ABB RAPID module: 93bc2229-db1b-41b8-8230-48410be7e35f-Module1.mod

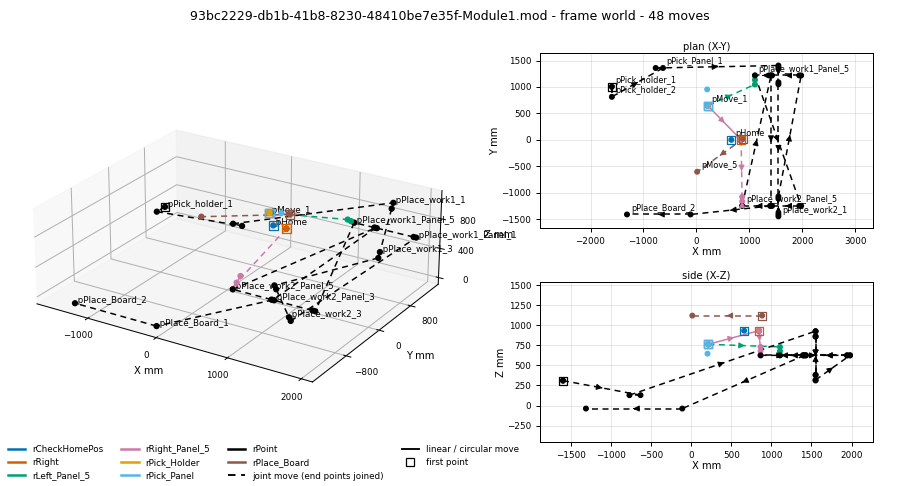
[picture p0: tool path of 93bc2229-db1b-41b8-8230-48410be7e35f-Module1.mod in frame world, 48 of 79 moves have a stored position in this frame; points joined in program order, loops and branches not executed]
MODULE Module1
    PERS tooldata Tool_Vacuum:=[TRUE,[[0,0.098,155.795],[1,0,0,0]],[5,[0,0,50],[1,0,0,0],0,0,0]];
	TASK PERS wobjdata Wobj_materials:=[FALSE,TRUE,"",[[-2196.81,858.538,-168],[1,0,0,0]],[[0,0,0],[1,0,0,0]]];
	TASK PERS wobjdata Wobj_Board:=[FALSE,TRUE,"",[[-2051.58,-1907.53,-168],[1,0,0,0]],[[0,0,0],[1,0,0,0]]];
	TASK PERS wobjdata Wobj_Left:=[FALSE,TRUE,"",[[802.356,885.126,-138],[0.872954,0.487803,0,0]],[[0,0,0],[1,0,0,0]]];
	TASK PERS wobjdata Wobj_Right:=[FALSE,TRUE,"",[[802.356,-1714.87,1162],[0.872954,-0.487803,0,0]],[[0,0,0],[1,0,0,0]]];
    PERS robtarget pHome:=[[661.17,-0.00,932.98],[3.16101E-08,-0.707107,-0.707107,-7.01508E-10],[-1,0,0,0],[9E+09,9E+09,9E+09,9E+09,9E+09,9E+09]];
    PERS robtarget pPick_holder_1:=[[600.00,145.65,477.91],[4.68845E-08,1.19209E-07,1,-2.94814E-08],[1,0,1,0],[9E+09,9E+09,9E+09,9E+09,9E+09,9E+09]];
    PERS robtarget pPick_holder_2:=[[600.00,-45.54,478.84],[7.08134E-08,4.45843E-09,1,-4.04558E-08],[1,0,1,0],[9E+09,9E+09,9E+09,9E+09,9E+09,9E+09]];
    PERS robtarget pPick_Panel_1:=[[1566.56,500.00,297.53],[2.60305E-09,0.707107,0.707107,-1.31181E-08],[1,0,2,0],[9E+09,9E+09,9E+09,9E+09,9E+09,9E+09]];
    PERS robtarget pPick_Panel_2:=[[1428.44,500.00,297.53],[3.82813E-09,0.707107,0.707107,-1.22165E-08],[1,0,2,0],[9E+09,9E+09,9E+09,9E+09,9E+09,9E+09]];
    PERS robtarget pPick_Holder_Move1{4,10}:=[[[[600,145.65,477.91],[4.68845E-8,1.19209E-7,1,-2.94814E-8],[1,0,1,0],[9E+9,9E+9,9E+9,9E+9,9E+9,9E+9]],[[600,245.65,477.91],[4.68845E-8,1.19209E-7,1,-2.94814E-8],[1,0,1,0],[9E+9,9E+9,9E+9,9E+9,9E+9,9E+9]],[[600,345.65,477.91],[4.68845E-8,1.19209E-7,1,-2.94814E-8],[1,0,1,0],[9E+9,9E+9,9E+9,9E+9,9E+9,9E+9]],[[600,445.65,477.91],[4.68845E-8,1.19209E-7,1,-2.94814E-8],[1,0,1,0],[9E+9,9E+9,9E+9,9E+9,9E+9,9E+9]],[[600,545.65,477.91],[4.68845E-8,1.19209E-7,1,-2.94814E-8],[1,0,1,0],[9E+9,9E+9,9E+9,9E+9,9E+9,9E+9]],[[600,645.65,477.91],[4.68845E-8,1.19209E-7,1,-2.94814E-8],[1,0,1,0],[9E+9,9E+9,9E+9,9E+9,9E+9,9E+9]],[[600,745.65,477.91],[4.68845E-8,1.19209E-7,1,-2.94814E-8],[1,0,1,0],[9E+9,9E+9,9E+9,9E+9,9E+9,9E+9]],[[600,845.65,477.91],[4.68845E-8,1.19209E-7,1,-2.94814E-8],[1,0,1,0],[9E+9,9E+9,9E+9,9E+9,9E+9,9E+9]],[[600,945.65,477.91],[4.68845E-8,1.19209E-7,1,-2.94814E-8],[1,0,1,0],[9E+9,9E+9,9E+9,9E+9,9E+9,9E+9]],[[600,1045.65,477.91],[4.68845E-8,1.19209E-7,1,-2.94814E-8],[1,0,1,0],[9E+9,9E+9,9E+9,9E+9,9E+9,9E+9]]],[[[600,145.65,357.91],[4.68845E-8,1.19209E-7,1,-2.94814E-8],[1,0,1,0],[9E+9,9E+9,9E+9,9E+9,9E+9,9E+9]],[[600,245.65,357.91],[4.68845E-8,1.19209E-7,1,-2.94814E-8],[1,0,1,0],[9E+9,9E+9,9E+9,9E+9,9E+9,9E+9]],[[600,345.65,357.91],[4.68845E-8,1.19209E-7,1,-2.94814E-8],[1,0,1,0],[9E+9,9E+9,9E+9,9E+9,9E+9,9E+9]],[[600,445.65,357.91],[4.68845E-8,1.19209E-7,1,-2.94814E-8],[1,0,1,0],[9E+9,9E+9,9E+9,9E+9,9E+9,9E+9]],[[600,545.65,357.91],[4.68845E-8,1.19209E-7,1,-2.94814E-8],[1,0,1,0],[9E+9,9E+9,9E+9,9E+9,9E+9,9E+9]],[[600,645.65,357.91],[4.68845E-8,1.19209E-7,1,-2.94814E-8],[1,0,1,0],[9E+9,9E+9,9E+9,9E+9,9E+9,9E+9]],[[600,745.65,357.91],[4.68845E-8,1.19209E-7,1,-2.94814E-8],[1,0,1,0],[9E+9,9E+9,9E+9,9E+9,9E+9,9E+9]],[[600,845.65,357.91],[4.68845E-8,1.19209E-7,1,-2.94814E-8],[1,0,1,0],[9E+9,9E+9,9E+9,9E+9,9E+9,9E+9]],[[600,945.65,357.91],[4.68845E-8,1.19209E-7,1,-2.94814E-8],[1,0,1,0],[9E+9,9E+9,9E+9,9E+9,9E+9,9E+9]],[[600,1045.65,357.91],[4.68845E-8,1.19209E-7,1,-2.94814E-8],[1,0,1,0],[9E+9,9E+9,9E+9,9E+9,9E+9,9E+9]]],[[[600,145.65,237.91],[4.68845E-8,1.19209E-7,1,-2.94814E-8],[1,0,1,0],[9E+9,9E+9,9E+9,9E+9,9E+9,9E+9]],[[600,245.65,237.91],[4.68845E-8,1.19209E-7,1,-2.94814E-8],[1,0,1,0],[9E+9,9E+9,9E+9,9E+9,9E+9,9E+9]],[[600,345.65,237.91],[4.68845E-8,1.19209E-7,1,-2.94814E-8],[1,0,1,0],[9E+9,9E+9,9E+9,9E+9,9E+9,9E+9]],[[600,445.65,237.91],[4.68845E-8,1.19209E-7,1,-2.94814E-8],[1,0,1,0],[9E+9,9E+9,9E+9,9E+9,9E+9,9E+9]],[[600,545.65,237.91],[4.68845E-8,1.19209E-7,1,-2.94814E-8],[1,0,1,0],[9E+9,9E+9,9E+9,9E+9,9E+9,9E+9]],[[600,645.65,237.91],[4.68845E-8,1.19209E-7,1,-2.94814E-8],[1,0,1,0],[9E+9,9E+9,9E+9,9E+9,9E+9,9E+9]],[[600,745.65,237.91],[4.68845E-8,1.19209E-7,1,-2.94814E-8],[1,0,1,0],[9E+9,9E+9,9E+9,9E+9,9E+9,9E+9]],[[600,845.65,237.91],[4.68845E-8,1.19209E-7,1,-2.94814E-8],[1,0,1,0],[9E+9,9E+9,9E+9,9E+9,9E+9,9E+9]],[[600,945.65,237.91],[4.68845E-8,1.19209E-7,1,-2.94814E-8],[1,0,1,0],[9E+9,9E+9,9E+9,9E+9,9E+9,9E+9]],[[600,1045.65,237.91],[4.68845E-8,1.19209E-7,1,-2.94814E-8],[1,0,1,0],[9E+9,9E+9,9E+9,9E+9,9E+9,9E+9]]],[[[600,145.65,117.91],[4.68845E-8,1.19209E-7,1,-2.94814E-8],[1,0,1,0],[9E+9,9E+9,9E+9,9E+9,9E+9,9E+9]],[[600,245.65,117.91],[4.68845E-8,1.19209E-7,1,-2.94814E-8],[1,0,1,0],[9E+9,9E+9,9E+9,9E+9,9E+9,9E+9]],[[600,345.65,117.91],[4.68845E-8,1.19209E-7,1,-2.94814E-8],[1,0,1,0],[9E+9,9E+9,9E+9,9E+9,9E+9,9E+9]],[[600,445.65,117.91],[4.68845E-8,1.19209E-7,1,-2.94814E-8],[1,0,1,0],[9E+9,9E+9,9E+9,9E+9,9E+9,9E+9]],[[600,545.65,117.91],[4.68845E-8,1.19209E-7,1,-2.94814E-8],[1,0,1,0],[9E+9,9E+9,9E+9,9E+9,9E+9,9E+9]],[[600,645.65,117.91],[4.68845E-8,1.19209E-7,1,-2.94814E-8],[1,0,1,0],[9E+9,9E+9,9E+9,9E+9,9E+9,9E+9]],[[600,745.65,117.91],[4.68845E-8,1.19209E-7,1,-2.94814E-8],[1,0,1,0],[9E+9,9E+9,9E+9,9E+9,9E+9,9E+9]],[[600,845.65,117.91],[4.68845E-8,1.19209E-7,1,-2.94814E-8],[1,0,1,0],[9E+9,9E+9,9E+9,9E+9,9E+9,9E+9]],[[600,945.65,117.91],[4.68845E-8,1.19209E-7,1,-2.94814E-8],[1,0,1,0],[9E+9,9E+9,9E+9,9E+9,9E+9,9E+9]],[[600,1045.65,117.91],[4.68845E-8,1.19209E-7,1,-2.94814E-8],[1,0,1,0],[9E+9,9E+9,9E+9,9E+9,9E+9,9E+9]]]];
    PERS robtarget pPick_Holder_Move2{4,10}:=[[[[600,-45.54,478.84],[7.08134E-8,4.45843E-9,1,-4.04558E-8],[1,0,1,0],[9E+9,9E+9,9E+9,9E+9,9E+9,9E+9]],[[600,54.46,478.84],[7.08134E-8,4.45843E-9,1,-4.04558E-8],[1,0,1,0],[9E+9,9E+9,9E+9,9E+9,9E+9,9E+9]],[[600,154.46,478.84],[7.08134E-8,4.45843E-9,1,-4.04558E-8],[1,0,1,0],[9E+9,9E+9,9E+9,9E+9,9E+9,9E+9]],[[600,254.46,478.84],[7.08134E-8,4.45843E-9,1,-4.04558E-8],[1,0,1,0],[9E+9,9E+9,9E+9,9E+9,9E+9,9E+9]],[[600,354.46,478.84],[7.08134E-8,4.45843E-9,1,-4.04558E-8],[1,0,1,0],[9E+9,9E+9,9E+9,9E+9,9E+9,9E+9]],[[600,454.46,478.84],[7.08134E-8,4.45843E-9,1,-4.04558E-8],[1,0,1,0],[9E+9,9E+9,9E+9,9E+9,9E+9,9E+9]],[[600,554.46,478.84],[7.08134E-8,4.45843E-9,1,-4.04558E-8],[1,0,1,0],[9E+9,9E+9,9E+9,9E+9,9E+9,9E+9]],[[600,654.46,478.84],[7.08134E-8,4.45843E-9,1,-4.04558E-8],[1,0,1,0],[9E+9,9E+9,9E+9,9E+9,9E+9,9E+9]],[[600,754.46,478.84],[7.08134E-8,4.45843E-9,1,-4.04558E-8],[1,0,1,0],[9E+9,9E+9,9E+9,9E+9,9E+9,9E+9]],[[600,854.46,478.84],[7.08134E-8,4.45843E-9,1,-4.04558E-8],[1,0,1,0],[9E+9,9E+9,9E+9,9E+9,9E+9,9E+9]]],[[[600,-45.54,358.84],[7.08134E-8,4.45843E-9,1,-4.04558E-8],[1,0,1,0],[9E+9,9E+9,9E+9,9E+9,9E+9,9E+9]],[[600,54.46,358.84],[7.08134E-8,4.45843E-9,1,-4.04558E-8],[1,0,1,0],[9E+9,9E+9,9E+9,9E+9,9E+9,9E+9]],[[600,154.46,358.84],[7.08134E-8,4.45843E-9,1,-4.04558E-8],[1,0,1,0],[9E+9,9E+9,9E+9,9E+9,9E+9,9E+9]],[[600,254.46,358.84],[7.08134E-8,4.45843E-9,1,-4.04558E-8],[1,0,1,0],[9E+9,9E+9,9E+9,9E+9,9E+9,9E+9]],[[600,354.46,358.84],[7.08134E-8,4.45843E-9,1,-4.04558E-8],[1,0,1,0],[9E+9,9E+9,9E+9,9E+9,9E+9,9E+9]],[[600,454.46,358.84],[7.08134E-8,4.45843E-9,1,-4.04558E-8],[1,0,1,0],[9E+9,9E+9,9E+9,9E+9,9E+9,9E+9]],[[600,554.46,358.84],[7.08134E-8,4.45843E-9,1,-4.04558E-8],[1,0,1,0],[9E+9,9E+9,9E+9,9E+9,9E+9,9E+9]],[[600,654.46,358.84],[7.08134E-8,4.45843E-9,1,-4.04558E-8],[1,0,1,0],[9E+9,9E+9,9E+9,9E+9,9E+9,9E+9]],[[600,754.46,358.84],[7.08134E-8,4.45843E-9,1,-4.04558E-8],[1,0,1,0],[9E+9,9E+9,9E+9,9E+9,9E+9,9E+9]],[[600,854.46,358.84],[7.08134E-8,4.45843E-9,1,-4.04558E-8],[1,0,1,0],[9E+9,9E+9,9E+9,9E+9,9E+9,9E+9]]],[[[600,-45.54,238.84],[7.08134E-8,4.45843E-9,1,-4.04558E-8],[1,0,1,0],[9E+9,9E+9,9E+9,9E+9,9E+9,9E+9]],[[600,54.46,238.84],[7.08134E-8,4.45843E-9,1,-4.04558E-8],[1,0,1,0],[9E+9,9E+9,9E+9,9E+9,9E+9,9E+9]],[[600,154.46,238.84],[7.08134E-8,4.45843E-9,1,-4.04558E-8],[1,0,1,0],[9E+9,9E+9,9E+9,9E+9,9E+9,9E+9]],[[600,254.46,238.84],[7.08134E-8,4.45843E-9,1,-4.04558E-8],[1,0,1,0],[9E+9,9E+9,9E+9,9E+9,9E+9,9E+9]],[[600,354.46,238.84],[7.08134E-8,4.45843E-9,1,-4.04558E-8],[1,0,1,0],[9E+9,9E+9,9E+9,9E+9,9E+9,9E+9]],[[600,454.46,238.84],[7.08134E-8,4.45843E-9,1,-4.04558E-8],[1,0,1,0],[9E+9,9E+9,9E+9,9E+9,9E+9,9E+9]],[[600,554.46,238.84],[7.08134E-8,4.45843E-9,1,-4.04558E-8],[1,0,1,0],[9E+9,9E+9,9E+9,9E+9,9E+9,9E+9]],[[600,654.46,238.84],[7.08134E-8,4.45843E-9,1,-4.04558E-8],[1,0,1,0],[9E+9,9E+9,9E+9,9E+9,9E+9,9E+9]],[[600,754.46,238.84],[7.08134E-8,4.45843E-9,1,-4.04558E-8],[1,0,1,0],[9E+9,9E+9,9E+9,9E+9,9E+9,9E+9]],[[600,854.46,238.84],[7.08134E-8,4.45843E-9,1,-4.04558E-8],[1,0,1,0],[9E+9,9E+9,9E+9,9E+9,9E+9,9E+9]]],[[[600,-45.54,118.84],[7.08134E-8,4.45843E-9,1,-4.04558E-8],[1,0,1,0],[9E+9,9E+9,9E+9,9E+9,9E+9,9E+9]],[[600,54.46,118.84],[7.08134E-8,4.45843E-9,1,-4.04558E-8],[1,0,1,0],[9E+9,9E+9,9E+9,9E+9,9E+9,9E+9]],[[600,154.46,118.84],[7.08134E-8,4.45843E-9,1,-4.04558E-8],[1,0,1,0],[9E+9,9E+9,9E+9,9E+9,9E+9,9E+9]],[[600,254.46,118.84],[7.08134E-8,4.45843E-9,1,-4.04558E-8],[1,0,1,0],[9E+9,9E+9,9E+9,9E+9,9E+9,9E+9]],[[600,354.46,118.84],[7.08134E-8,4.45843E-9,1,-4.04558E-8],[1,0,1,0],[9E+9,9E+9,9E+9,9E+9,9E+9,9E+9]],[[600,454.46,118.84],[7.08134E-8,4.45843E-9,1,-4.04558E-8],[1,0,1,0],[9E+9,9E+9,9E+9,9E+9,9E+9,9E+9]],[[600,554.46,118.84],[7.08134E-8,4.45843E-9,1,-4.04558E-8],[1,0,1,0],[9E+9,9E+9,9E+9,9E+9,9E+9,9E+9]],[[600,654.46,118.84],[7.08134E-8,4.45843E-9,1,-4.04558E-8],[1,0,1,0],[9E+9,9E+9,9E+9,9E+9,9E+9,9E+9]],[[600,754.46,118.84],[7.08134E-8,4.45843E-9,1,-4.04558E-8],[1,0,1,0],[9E+9,9E+9,9E+9,9E+9,9E+9,9E+9]],[[600,854.46,118.84],[7.08134E-8,4.45843E-9,1,-4.04558E-8],[1,0,1,0],[9E+9,9E+9,9E+9,9E+9,9E+9,9E+9]]]];
    PERS robtarget pPick_Panel_Move1{20,5}:=[[[[1566.56,500,297.53],[2.60305E-9,0.707107,0.707107,-1.31181E-8],[1,0,2,0],[9E+9,9E+9,9E+9,9E+9,9E+9,9E+9]],[[1766.56,500,297.53],[2.60305E-9,0.707107,0.707107,-1.31181E-8],[1,0,2,0],[9E+9,9E+9,9E+9,9E+9,9E+9,9E+9]],[[1966.56,500,297.53],[2.60305E-9,0.707107,0.707107,-1.31181E-8],[1,0,2,0],[9E+9,9E+9,9E+9,9E+9,9E+9,9E+9]],[[2166.56,500,297.53],[2.60305E-9,0.707107,0.707107,-1.31181E-8],[1,0,2,0],[9E+9,9E+9,9E+9,9E+9,9E+9,9E+9]],[[2366.56,500,297.53],[2.60305E-9,0.707107,0.707107,-1.31181E-8],[1,0,2,0],[9E+9,9E+9,9E+9,9E+9,9E+9,9E+9]]],[[[1566.56,500,282.53],[2.60305E-9,0.707107,0.707107,-1.31181E-8],[1,0,2,0],[9E+9,9E+9,9E+9,9E+9,9E+9,9E+9]],[[1766.56,500,282.53],[2.60305E-9,0.707107,0.707107,-1.31181E-8],[1,0,2,0],[9E+9,9E+9,9E+9,9E+9,9E+9,9E+9]],[[1966.56,500,282.53],[2.60305E-9,0.707107,0.707107,-1.31181E-8],[1,0,2,0],[9E+9,9E+9,9E+9,9E+9,9E+9,9E+9]],[[2166.56,500,282.53],[2.60305E-9,0.707107,0.707107,-1.31181E-8],[1,0,2,0],[9E+9,9E+9,9E+9,9E+9,9E+9,9E+9]],[[2366.56,500,282.53],[2.60305E-9,0.707107,0.707107,-1.31181E-8],[1,0,2,0],[9E+9,9E+9,9E+9,9E+9,9E+9,9E+9]]],[[[1566.56,500,267.53],[2.60305E-9,0.707107,0.707107,-1.31181E-8],[1,0,2,0],[9E+9,9E+9,9E+9,9E+9,9E+9,9E+9]],[[1766.56,500,267.53],[2.60305E-9,0.707107,0.707107,-1.31181E-8],[1,0,2,0],[9E+9,9E+9,9E+9,9E+9,9E+9,9E+9]],[[1966.56,500,267.53],[2.60305E-9,0.707107,0.707107,-1.31181E-8],[1,0,2,0],[9E+9,9E+9,9E+9,9E+9,9E+9,9E+9]],[[2166.56,500,267.53],[2.60305E-9,0.707107,0.707107,-1.31181E-8],[1,0,2,0],[9E+9,9E+9,9E+9,9E+9,9E+9,9E+9]],[[2366.56,500,267.53],[2.60305E-9,0.707107,0.707107,-1.31181E-8],[1,0,2,0],[9E+9,9E+9,9E+9,9E+9,9E+9,9E+9]]],[[[1566.56,500,252.53],[2.60305E-9,0.707107,0.707107,-1.31181E-8],[1,0,2,0],[9E+9,9E+9,9E+9,9E+9,9E+9,9E+9]],[[1766.56,500,252.53],[2.60305E-9,0.707107,0.707107,-1.31181E-8],[1,0,2,0],[9E+9,9E+9,9E+9,9E+9,9E+9,9E+9]],[[1966.56,500,252.53],[2.60305E-9,0.707107,0.707107,-1.31181E-8],[1,0,2,0],[9E+9,9E+9,9E+9,9E+9,9E+9,9E+9]],[[2166.56,500,252.53],[2.60305E-9,0.707107,0.707107,-1.31181E-8],[1,0,2,0],[9E+9,9E+9,9E+9,9E+9,9E+9,9E+9]],[[2366.56,500,252.53],[2.60305E-9,0.707107,0.707107,-1.31181E-8],[1,0,2,0],[9E+9,9E+9,9E+9,9E+9,9E+9,9E+9]]],[[[1566.56,500,237.53],[2.60305E-9,0.707107,0.707107,-1.31181E-8],[1,0,2,0],[9E+9,9E+9,9E+9,9E+9,9E+9,9E+9]],[[1766.56,500,237.53],[2.60305E-9,0.707107,0.707107,-1.31181E-8],[1,0,2,0],[9E+9,9E+9,9E+9,9E+9,9E+9,9E+9]],[[1966.56,500,237.53],[2.60305E-9,0.707107,0.707107,-1.31181E-8],[1,0,2,0],[9E+9,9E+9,9E+9,9E+9,9E+9,9E+9]],[[2166.56,500,237.53],[2.60305E-9,0.707107,0.707107,-1.31181E-8],[1,0,2,0],[9E+9,9E+9,9E+9,9E+9,9E+9,9E+9]],[[2366.56,500,237.53],[2.60305E-9,0.707107,0.707107,-1.31181E-8],[1,0,2,0],[9E+9,9E+9,9E+9,9E+9,9E+9,9E+9]]],[[[1566.56,500,222.53],[2.60305E-9,0.707107,0.707107,-1.31181E-8],[1,0,2,0],[9E+9,9E+9,9E+9,9E+9,9E+9,9E+9]],[[1766.56,500,222.53],[2.60305E-9,0.707107,0.707107,-1.31181E-8],[1,0,2,0],[9E+9,9E+9,9E+9,9E+9,9E+9,9E+9]],[[1966.56,500,222.53],[2.60305E-9,0.707107,0.707107,-1.31181E-8],[1,0,2,0],[9E+9,9E+9,9E+9,9E+9,9E+9,9E+9]],[[2166.56,500,222.53],[2.60305E-9,0.707107,0.707107,-1.31181E-8],[1,0,2,0],[9E+9,9E+9,9E+9,9E+9,9E+9,9E+9]],[[2366.56,500,222.53],[2.60305E-9,0.707107,0.707107,-1.31181E-8],[1,0,2,0],[9E+9,9E+9,9E+9,9E+9,9E+9,9E+9]]],[[[1566.56,500,207.53],[2.60305E-9,0.707107,0.707107,-1.31181E-8],[1,0,2,0],[9E+9,9E+9,9E+9,9E+9,9E+9,9E+9]],[[1766.56,500,207.53],[2.60305E-9,0.707107,0.707107,-1.31181E-8],[1,0,2,0],[9E+9,9E+9,9E+9,9E+9,9E+9,9E+9]],[[1966.56,500,207.53],[2.60305E-9,0.707107,0.707107,-1.31181E-8],[1,0,2,0],[9E+9,9E+9,9E+9,9E+9,9E+9,9E+9]],[[2166.56,500,207.53],[2.60305E-9,0.707107,0.707107,-1.31181E-8],[1,0,2,0],[9E+9,9E+9,9E+9,9E+9,9E+9,9E+9]],[[2366.56,500,207.53],[2.60305E-9,0.707107,0.707107,-1.31181E-8],[1,0,2,0],[9E+9,9E+9,9E+9,9E+9,9E+9,9E+9]]],[[[1566.56,500,192.53],[2.60305E-9,0.707107,0.707107,-1.31181E-8],[1,0,2,0],[9E+9,9E+9,9E+9,9E+9,9E+9,9E+9]],[[1766.56,500,192.53],[2.60305E-9,0.707107,0.707107,-1.31181E-8],[1,0,2,0],[9E+9,9E+9,9E+9,9E+9,9E+9,9E+9]],[[1966.56,500,192.53],[2.60305E-9,0.707107,0.707107,-1.31181E-8],[1,0,2,0],[9E+9,9E+9,9E+9,9E+9,9E+9,9E+9]],[[2166.56,500,192.53],[2.60305E-9,0.707107,0.707107,-1.31181E-8],[1,0,2,0],[9E+9,9E+9,9E+9,9E+9,9E+9,9E+9]],[[2366.56,500,192.53],[2.60305E-9,0.707107,0.707107,-1.31181E-8],[1,0,2,0],[9E+9,9E+9,9E+9,9E+9,9E+9,9E+9]]],[[[1566.56,500,177.53],[2.60305E-9,0.707107,0.707107,-1.31181E-8],[1,0,2,0],[9E+9,9E+9,9E+9,9E+9,9E+9,9E+9]],[[1766.56,500,177.53],[2.60305E-9,0.707107,0.707107,-1.31181E-8],[1,0,2,0],[9E+9,9E+9,9E+9,9E+9,9E+9,9E+9]],[[1966.56,500,177.53],[2.60305E-9,0.707107,0.707107,-1.31181E-8],[1,0,2,0],[9E+9,9E+9,9E+9,9E+9,9E+9,9E+9]],[[2166.56,500,177.53],[2.60305E-9,0.707107,0.707107,-1.31181E-8],[1,0,2,0],[9E+9,9E+9,9E+9,9E+9,9E+9,9E+9]],[[2366.56,500,177.53],[2.60305E-9,0.707107,0.707107,-1.31181E-8],[1,0,2,0],[9E+9,9E+9,9E+9,9E+9,9E+9,9E+9]]],[[[1566.56,500,162.53],[2.60305E-9,0.707107,0.707107,-1.31181E-8],[1,0,2,0],[9E+9,9E+9,9E+9,9E+9,9E+9,9E+9]],[[1766.56,500,162.53],[2.60305E-9,0.707107,0.707107,-1.31181E-8],[1,0,2,0],[9E+9,9E+9,9E+9,9E+9,9E+9,9E+9]],[[1966.56,500,162.53],[2.60305E-9,0.707107,0.707107,-1.31181E-8],[1,0,2,0],[9E+9,9E+9,9E+9,9E+9,9E+9,9E+9]],[[2166.56,500,162.53],[2.60305E-9,0.707107,0.707107,-1.31181E-8],[1,0,2,0],[9E+9,9E+9,9E+9,9E+9,9E+9,9E+9]],[[2366.56,500,162.53],[2.60305E-9,0.707107,0.707107,-1.31181E-8],[1,0,2,0],[9E+9,9E+9,9E+9,9E+9,9E+9,9E+9]]],[[[1566.56,500,147.53],[2.60305E-9,0.707107,0.707107,-1.31181E-8],[1,0,2,0],[9E+9,9E+9,9E+9,9E+9,9E+9,9E+9]],[[1766.56,500,147.53],[2.60305E-9,0.707107,0.707107,-1.31181E-8],[1,0,2,0],[9E+9,9E+9,9E+9,9E+9,9E+9,9E+9]],[[1966.56,500,147.53],[2.60305E-9,0.707107,0.707107,-1.31181E-8],[1,0,2,0],[9E+9,9E+9,9E+9,9E+9,9E+9,9E+9]],[[2166.56,500,147.53],[2.60305E-9,0.707107,0.707107,-1.31181E-8],[1,0,2,0],[9E+9,9E+9,9E+9,9E+9,9E+9,9E+9]],[[2366.56,500,147.53],[2.60305E-9,0.707107,0.707107,-1.31181E-8],[1,0,2,0],[9E+9,9E+9,9E+9,9E+9,9E+9,9E+9]]],[[[1566.56,500,132.53],[2.60305E-9,0.707107,0.707107,-1.31181E-8],[1,0,2,0],[9E+9,9E+9,9E+9,9E+9,9E+9,9E+9]],[[1766.56,500,132.53],[2.60305E-9,0.707107,0.707107,-1.31181E-8],[1,0,2,0],[9E+9,9E+9,9E+9,9E+9,9E+9,9E+9]],[[1966.56,500,132.53],[2.60305E-9,0.707107,0.707107,-1.31181E-8],[1,0,2,0],[9E+9,9E+9,9E+9,9E+9,9E+9,9E+9]],[[2166.56,500,132.53],[2.60305E-9,0.707107,0.707107,-1.31181E-8],[1,0,2,0],[9E+9,9E+9,9E+9,9E+9,9E+9,9E+9]],[[2366.56,500,132.53],[2.60305E-9,0.707107,0.707107,-1.31181E-8],[1,0,2,0],[9E+9,9E+9,9E+9,9E+9,9E+9,9E+9]]],[[[1566.56,500,117.53],[2.60305E-9,0.707107,0.707107,-1.31181E-8],[1,0,2,0],[9E+9,9E+9,9E+9,9E+9,9E+9,9E+9]],[[1766.56,500,117.53],[2.60305E-9,0.707107,0.707107,-1.31181E-8],[1,0,2,0],[9E+9,9E+9,9E+9,9E+9,9E+9,9E+9]],[[1966.56,500,117.53],[2.60305E-9,0.707107,0.707107,-1.31181E-8],[1,0,2,0],[9E+9,9E+9,9E+9,9E+9,9E+9,9E+9]],[[2166.56,500,117.53],[2.60305E-9,0.707107,0.707107,-1.31181E-8],[1,0,2,0],[9E+9,9E+9,9E+9,9E+9,9E+9,9E+9]],[[2366.56,500,117.53],[2.60305E-9,0.707107,0.707107,-1.31181E-8],[1,0,2,0],[9E+9,9E+9,9E+9,9E+9,9E+9,9E+9]]],[[[1566.56,500,102.53],[2.60305E-9,0.707107,0.707107,-1.31181E-8],[1,0,2,0],[9E+9,9E+9,9E+9,9E+9,9E+9,9E+9]],[[1766.56,500,102.53],[2.60305E-9,0.707107,0.707107,-1.31181E-8],[1,0,2,0],[9E+9,9E+9,9E+9,9E+9,9E+9,9E+9]],[[1966.56,500,102.53],[2.60305E-9,0.707107,0.707107,-1.31181E-8],[1,0,2,0],[9E+9,9E+9,9E+9,9E+9,9E+9,9E+9]],[[2166.56,500,102.53],[2.60305E-9,0.707107,0.707107,-1.31181E-8],[1,0,2,0],[9E+9,9E+9,9E+9,9E+9,9E+9,9E+9]],[[2366.56,500,102.53],[2.60305E-9,0.707107,0.707107,-1.31181E-8],[1,0,2,0],[9E+9,9E+9,9E+9,9E+9,9E+9,9E+9]]],[[[1566.56,500,87.53],[2.60305E-9,0.707107,0.707107,-1.31181E-8],[1,0,2,0],[9E+9,9E+9,9E+9,9E+9,9E+9,9E+9]],[[1766.56,500,87.53],[2.60305E-9,0.707107,0.707107,-1.31181E-8],[1,0,2,0],[9E+9,9E+9,9E+9,9E+9,9E+9,9E+9]],[[1966.56,500,87.53],[2.60305E-9,0.707107,0.707107,-1.31181E-8],[1,0,2,0],[9E+9,9E+9,9E+9,9E+9,9E+9,9E+9]],[[2166.56,500,87.53],[2.60305E-9,0.707107,0.707107,-1.31181E-8],[1,0,2,0],[9E+9,9E+9,9E+9,9E+9,9E+9,9E+9]],[[2366.56,500,87.53],[2.60305E-9,0.707107,0.707107,-1.31181E-8],[1,0,2,0],[9E+9,9E+9,9E+9,9E+9,9E+9,9E+9]]],[[[1566.56,500,72.53],[2.60305E-9,0.707107,0.707107,-1.31181E-8],[1,0,2,0],[9E+9,9E+9,9E+9,9E+9,9E+9,9E+9]],[[1766.56,500,72.53],[2.60305E-9,0.707107,0.707107,-1.31181E-8],[1,0,2,0],[9E+9,9E+9,9E+9,9E+9,9E+9,9E+9]],[[1966.56,500,72.53],[2.60305E-9,0.707107,0.707107,-1.31181E-8],[1,0,2,0],[9E+9,9E+9,9E+9,9E+9,9E+9,9E+9]],[[2166.56,500,72.53],[2.60305E-9,0.707107,0.707107,-1.31181E-8],[1,0,2,0],[9E+9,9E+9,9E+9,9E+9,9E+9,9E+9]],[[2366.56,500,72.53],[2.60305E-9,0.707107,0.707107,-1.31181E-8],[1,0,2,0],[9E+9,9E+9,9E+9,9E+9,9E+9,9E+9]]],[[[1566.56,500,57.53],[2.60305E-9,0.707107,0.707107,-1.31181E-8],[1,0,2,0],[9E+9,9E+9,9E+9,9E+9,9E+9,9E+9]],[[1766.56,500,57.53],[2.60305E-9,0.707107,0.707107,-1.31181E-8],[1,0,2,0],[9E+9,9E+9,9E+9,9E+9,9E+9,9E+9]],[[1966.56,500,57.53],[2.60305E-9,0.707107,0.707107,-1.31181E-8],[1,0,2,0],[9E+9,9E+9,9E+9,9E+9,9E+9,9E+9]],[[2166.56,500,57.53],[2.60305E-9,0.707107,0.707107,-1.31181E-8],[1,0,2,0],[9E+9,9E+9,9E+9,9E+9,9E+9,9E+9]],[[2366.56,500,57.53],[2.60305E-9,0.707107,0.707107,-1.31181E-8],[1,0,2,0],[9E+9,9E+9,9E+9,9E+9,9E+9,9E+9]]],[[[1566.56,500,42.53],[2.60305E-9,0.707107,0.707107,-1.31181E-8],[1,0,2,0],[9E+9,9E+9,9E+9,9E+9,9E+9,9E+9]],[[1766.56,500,42.53],[2.60305E-9,0.707107,0.707107,-1.31181E-8],[1,0,2,0],[9E+9,9E+9,9E+9,9E+9,9E+9,9E+9]],[[1966.56,500,42.53],[2.60305E-9,0.707107,0.707107,-1.31181E-8],[1,0,2,0],[9E+9,9E+9,9E+9,9E+9,9E+9,9E+9]],[[2166.56,500,42.53],[2.60305E-9,0.707107,0.707107,-1.31181E-8],[1,0,2,0],[9E+9,9E+9,9E+9,9E+9,9E+9,9E+9]],[[2366.56,500,42.53],[2.60305E-9,0.707107,0.707107,-1.31181E-8],[1,0,2,0],[9E+9,9E+9,9E+9,9E+9,9E+9,9E+9]]],[[[1566.56,500,27.53],[2.60305E-9,0.707107,0.707107,-1.31181E-8],[1,0,2,0],[9E+9,9E+9,9E+9,9E+9,9E+9,9E+9]],[[1766.56,500,27.53],[2.60305E-9,0.707107,0.707107,-1.31181E-8],[1,0,2,0],[9E+9,9E+9,9E+9,9E+9,9E+9,9E+9]],[[1966.56,500,27.53],[2.60305E-9,0.707107,0.707107,-1.31181E-8],[1,0,2,0],[9E+9,9E+9,9E+9,9E+9,9E+9,9E+9]],[[2166.56,500,27.53],[2.60305E-9,0.707107,0.707107,-1.31181E-8],[1,0,2,0],[9E+9,9E+9,9E+9,9E+9,9E+9,9E+9]],[[2366.56,500,27.53],[2.60305E-9,0.707107,0.707107,-1.31181E-8],[1,0,2,0],[9E+9,9E+9,9E+9,9E+9,9E+9,9E+9]]],[[[1566.56,500,12.53],[2.60305E-9,0.707107,0.707107,-1.31181E-8],[1,0,2,0],[9E+9,9E+9,9E+9,9E+9,9E+9,9E+9]],[[1766.56,500,12.53],[2.60305E-9,0.707107,0.707107,-1.31181E-8],[1,0,2,0],[9E+9,9E+9,9E+9,9E+9,9E+9,9E+9]],[[1966.56,500,12.53],[2.60305E-9,0.707107,0.707107,-1.31181E-8],[1,0,2,0],[9E+9,9E+9,9E+9,9E+9,9E+9,9E+9]],[[2166.56,500,12.53],[2.60305E-9,0.707107,0.707107,-1.31181E-8],[1,0,2,0],[9E+9,9E+9,9E+9,9E+9,9E+9,9E+9]],[[2366.56,500,12.53],[2.60305E-9,0.707107,0.707107,-1.31181E-8],[1,0,2,0],[9E+9,9E+9,9E+9,9E+9,9E+9,9E+9]]]];
    PERS robtarget pPick_Panel_Move2{20,5}:=[[[[1428.44,500,297.53],[3.82813E-9,0.707107,0.707107,-1.22165E-8],[1,0,2,0],[9E+9,9E+9,9E+9,9E+9,9E+9,9E+9]],[[1628.44,500,297.53],[3.82813E-9,0.707107,0.707107,-1.22165E-8],[1,0,2,0],[9E+9,9E+9,9E+9,9E+9,9E+9,9E+9]],[[1828.44,500,297.53],[3.82813E-9,0.707107,0.707107,-1.22165E-8],[1,0,2,0],[9E+9,9E+9,9E+9,9E+9,9E+9,9E+9]],[[2028.44,500,297.53],[3.82813E-9,0.707107,0.707107,-1.22165E-8],[1,0,2,0],[9E+9,9E+9,9E+9,9E+9,9E+9,9E+9]],[[2228.44,500,297.53],[3.82813E-9,0.707107,0.707107,-1.22165E-8],[1,0,2,0],[9E+9,9E+9,9E+9,9E+9,9E+9,9E+9]]],[[[1428.44,500,282.53],[3.82813E-9,0.707107,0.707107,-1.22165E-8],[1,0,2,0],[9E+9,9E+9,9E+9,9E+9,9E+9,9E+9]],[[1628.44,500,282.53],[3.82813E-9,0.707107,0.707107,-1.22165E-8],[1,0,2,0],[9E+9,9E+9,9E+9,9E+9,9E+9,9E+9]],[[1828.44,500,282.53],[3.82813E-9,0.707107,0.707107,-1.22165E-8],[1,0,2,0],[9E+9,9E+9,9E+9,9E+9,9E+9,9E+9]],[[2028.44,500,282.53],[3.82813E-9,0.707107,0.707107,-1.22165E-8],[1,0,2,0],[9E+9,9E+9,9E+9,9E+9,9E+9,9E+9]],[[2228.44,500,282.53],[3.82813E-9,0.707107,0.707107,-1.22165E-8],[1,0,2,0],[9E+9,9E+9,9E+9,9E+9,9E+9,9E+9]]],[[[1428.44,500,267.53],[3.82813E-9,0.707107,0.707107,-1.22165E-8],[1,0,2,0],[9E+9,9E+9,9E+9,9E+9,9E+9,9E+9]],[[1628.44,500,267.53],[3.82813E-9,0.707107,0.707107,-1.22165E-8],[1,0,2,0],[9E+9,9E+9,9E+9,9E+9,9E+9,9E+9]],[[1828.44,500,267.53],[3.82813E-9,0.707107,0.707107,-1.22165E-8],[1,0,2,0],[9E+9,9E+9,9E+9,9E+9,9E+9,9E+9]],[[2028.44,500,267.53],[3.82813E-9,0.707107,0.707107,-1.22165E-8],[1,0,2,0],[9E+9,9E+9,9E+9,9E+9,9E+9,9E+9]],[[2228.44,500,267.53],[3.82813E-9,0.707107,0.707107,-1.22165E-8],[1,0,2,0],[9E+9,9E+9,9E+9,9E+9,9E+9,9E+9]]],[[[1428.44,500,252.53],[3.82813E-9,0.707107,0.707107,-1.22165E-8],[1,0,2,0],[9E+9,9E+9,9E+9,9E+9,9E+9,9E+9]],[[1628.44,500,252.53],[3.82813E-9,0.707107,0.707107,-1.22165E-8],[1,0,2,0],[9E+9,9E+9,9E+9,9E+9,9E+9,9E+9]],[[1828.44,500,252.53],[3.82813E-9,0.707107,0.707107,-1.22165E-8],[1,0,2,0],[9E+9,9E+9,9E+9,9E+9,9E+9,9E+9]],[[2028.44,500,252.53],[3.82813E-9,0.707107,0.707107,-1.22165E-8],[1,0,2,0],[9E+9,9E+9,9E+9,9E+9,9E+9,9E+9]],[[2228.44,500,252.53],[3.82813E-9,0.707107,0.707107,-1.22165E-8],[1,0,2,0],[9E+9,9E+9,9E+9,9E+9,9E+9,9E+9]]],[[[1428.44,500,237.53],[3.82813E-9,0.707107,0.707107,-1.22165E-8],[1,0,2,0],[9E+9,9E+9,9E+9,9E+9,9E+9,9E+9]],[[1628.44,500,237.53],[3.82813E-9,0.707107,0.707107,-1.22165E-8],[1,0,2,0],[9E+9,9E+9,9E+9,9E+9,9E+9,9E+9]],[[1828.44,500,237.53],[3.82813E-9,0.707107,0.707107,-1.22165E-8],[1,0,2,0],[9E+9,9E+9,9E+9,9E+9,9E+9,9E+9]],[[2028.44,500,237.53],[3.82813E-9,0.707107,0.707107,-1.22165E-8],[1,0,2,0],[9E+9,9E+9,9E+9,9E+9,9E+9,9E+9]],[[2228.44,500,237.53],[3.82813E-9,0.707107,0.707107,-1.22165E-8],[1,0,2,0],[9E+9,9E+9,9E+9,9E+9,9E+9,9E+9]]],[[[1428.44,500,222.53],[3.82813E-9,0.707107,0.707107,-1.22165E-8],[1,0,2,0],[9E+9,9E+9,9E+9,9E+9,9E+9,9E+9]],[[1628.44,500,222.53],[3.82813E-9,0.707107,0.707107,-1.22165E-8],[1,0,2,0],[9E+9,9E+9,9E+9,9E+9,9E+9,9E+9]],[[1828.44,500,222.53],[3.82813E-9,0.707107,0.707107,-1.22165E-8],[1,0,2,0],[9E+9,9E+9,9E+9,9E+9,9E+9,9E+9]],[[2028.44,500,222.53],[3.82813E-9,0.707107,0.707107,-1.22165E-8],[1,0,2,0],[9E+9,9E+9,9E+9,9E+9,9E+9,9E+9]],[[2228.44,500,222.53],[3.82813E-9,0.707107,0.707107,-1.22165E-8],[1,0,2,0],[9E+9,9E+9,9E+9,9E+9,9E+9,9E+9]]],[[[1428.44,500,207.53],[3.82813E-9,0.707107,0.707107,-1.22165E-8],[1,0,2,0],[9E+9,9E+9,9E+9,9E+9,9E+9,9E+9]],[[1628.44,500,207.53],[3.82813E-9,0.707107,0.707107,-1.22165E-8],[1,0,2,0],[9E+9,9E+9,9E+9,9E+9,9E+9,9E+9]],[[1828.44,500,207.53],[3.82813E-9,0.707107,0.707107,-1.22165E-8],[1,0,2,0],[9E+9,9E+9,9E+9,9E+9,9E+9,9E+9]],[[2028.44,500,207.53],[3.82813E-9,0.707107,0.707107,-1.22165E-8],[1,0,2,0],[9E+9,9E+9,9E+9,9E+9,9E+9,9E+9]],[[2228.44,500,207.53],[3.82813E-9,0.707107,0.707107,-1.22165E-8],[1,0,2,0],[9E+9,9E+9,9E+9,9E+9,9E+9,9E+9]]],[[[1428.44,500,192.53],[3.82813E-9,0.707107,0.707107,-1.22165E-8],[1,0,2,0],[9E+9,9E+9,9E+9,9E+9,9E+9,9E+9]],[[1628.44,500,192.53],[3.82813E-9,0.707107,0.707107,-1.22165E-8],[1,0,2,0],[9E+9,9E+9,9E+9,9E+9,9E+9,9E+9]],[[1828.44,500,192.53],[3.82813E-9,0.707107,0.707107,-1.22165E-8],[1,0,2,0],[9E+9,9E+9,9E+9,9E+9,9E+9,9E+9]],[[2028.44,500,192.53],[3.82813E-9,0.707107,0.707107,-1.22165E-8],[1,0,2,0],[9E+9,9E+9,9E+9,9E+9,9E+9,9E+9]],[[2228.44,500,192.53],[3.82813E-9,0.707107,0.707107,-1.22165E-8],[1,0,2,0],[9E+9,9E+9,9E+9,9E+9,9E+9,9E+9]]],[[[1428.44,500,177.53],[3.82813E-9,0.707107,0.707107,-1.22165E-8],[1,0,2,0],[9E+9,9E+9,9E+9,9E+9,9E+9,9E+9]],[[1628.44,500,177.53],[3.82813E-9,0.707107,0.707107,-1.22165E-8],[1,0,2,0],[9E+9,9E+9,9E+9,9E+9,9E+9,9E+9]],[[1828.44,500,177.53],[3.82813E-9,0.707107,0.707107,-1.22165E-8],[1,0,2,0],[9E+9,9E+9,9E+9,9E+9,9E+9,9E+9]],[[2028.44,500,177.53],[3.82813E-9,0.707107,0.707107,-1.22165E-8],[1,0,2,0],[9E+9,9E+9,9E+9,9E+9,9E+9,9E+9]],[[2228.44,500,177.53],[3.82813E-9,0.707107,0.707107,-1.22165E-8],[1,0,2,0],[9E+9,9E+9,9E+9,9E+9,9E+9,9E+9]]],[[[1428.44,500,162.53],[3.82813E-9,0.707107,0.707107,-1.22165E-8],[1,0,2,0],[9E+9,9E+9,9E+9,9E+9,9E+9,9E+9]],[[1628.44,500,162.53],[3.82813E-9,0.707107,0.707107,-1.22165E-8],[1,0,2,0],[9E+9,9E+9,9E+9,9E+9,9E+9,9E+9]],[[1828.44,500,162.53],[3.82813E-9,0.707107,0.707107,-1.22165E-8],[1,0,2,0],[9E+9,9E+9,9E+9,9E+9,9E+9,9E+9]],[[2028.44,500,162.53],[3.82813E-9,0.707107,0.707107,-1.22165E-8],[1,0,2,0],[9E+9,9E+9,9E+9,9E+9,9E+9,9E+9]],[[2228.44,500,162.53],[3.82813E-9,0.707107,0.707107,-1.22165E-8],[1,0,2,0],[9E+9,9E+9,9E+9,9E+9,9E+9,9E+9]]],[[[1428.44,500,147.53],[3.82813E-9,0.707107,0.707107,-1.22165E-8],[1,0,2,0],[9E+9,9E+9,9E+9,9E+9,9E+9,9E+9]],[[1628.44,500,147.53],[3.82813E-9,0.707107,0.707107,-1.22165E-8],[1,0,2,0],[9E+9,9E+9,9E+9,9E+9,9E+9,9E+9]],[[1828.44,500,147.53],[3.82813E-9,0.707107,0.707107,-1.22165E-8],[1,0,2,0],[9E+9,9E+9,9E+9,9E+9,9E+9,9E+9]],[[2028.44,500,147.53],[3.82813E-9,0.707107,0.707107,-1.22165E-8],[1,0,2,0],[9E+9,9E+9,9E+9,9E+9,9E+9,9E+9]],[[2228.44,500,147.53],[3.82813E-9,0.707107,0.707107,-1.22165E-8],[1,0,2,0],[9E+9,9E+9,9E+9,9E+9,9E+9,9E+9]]],[[[1428.44,500,132.53],[3.82813E-9,0.707107,0.707107,-1.22165E-8],[1,0,2,0],[9E+9,9E+9,9E+9,9E+9,9E+9,9E+9]],[[1628.44,500,132.53],[3.82813E-9,0.707107,0.707107,-1.22165E-8],[1,0,2,0],[9E+9,9E+9,9E+9,9E+9,9E+9,9E+9]],[[1828.44,500,132.53],[3.82813E-9,0.707107,0.707107,-1.22165E-8],[1,0,2,0],[9E+9,9E+9,9E+9,9E+9,9E+9,9E+9]],[[2028.44,500,132.53],[3.82813E-9,0.707107,0.707107,-1.22165E-8],[1,0,2,0],[9E+9,9E+9,9E+9,9E+9,9E+9,9E+9]],[[2228.44,500,132.53],[3.82813E-9,0.707107,0.707107,-1.22165E-8],[1,0,2,0],[9E+9,9E+9,9E+9,9E+9,9E+9,9E+9]]],[[[1428.44,500,117.53],[3.82813E-9,0.707107,0.707107,-1.22165E-8],[1,0,2,0],[9E+9,9E+9,9E+9,9E+9,9E+9,9E+9]],[[1628.44,500,117.53],[3.82813E-9,0.707107,0.707107,-1.22165E-8],[1,0,2,0],[9E+9,9E+9,9E+9,9E+9,9E+9,9E+9]],[[1828.44,500,117.53],[3.82813E-9,0.707107,0.707107,-1.22165E-8],[1,0,2,0],[9E+9,9E+9,9E+9,9E+9,9E+9,9E+9]],[[2028.44,500,117.53],[3.82813E-9,0.707107,0.707107,-1.22165E-8],[1,0,2,0],[9E+9,9E+9,9E+9,9E+9,9E+9,9E+9]],[[2228.44,500,117.53],[3.82813E-9,0.707107,0.707107,-1.22165E-8],[1,0,2,0],[9E+9,9E+9,9E+9,9E+9,9E+9,9E+9]]],[[[1428.44,500,102.53],[3.82813E-9,0.707107,0.707107,-1.22165E-8],[1,0,2,0],[9E+9,9E+9,9E+9,9E+9,9E+9,9E+9]],[[1628.44,500,102.53],[3.82813E-9,0.707107,0.707107,-1.22165E-8],[1,0,2,0],[9E+9,9E+9,9E+9,9E+9,9E+9,9E+9]],[[1828.44,500,102.53],[3.82813E-9,0.707107,0.707107,-1.22165E-8],[1,0,2,0],[9E+9,9E+9,9E+9,9E+9,9E+9,9E+9]],[[2028.44,500,102.53],[3.82813E-9,0.707107,0.707107,-1.22165E-8],[1,0,2,0],[9E+9,9E+9,9E+9,9E+9,9E+9,9E+9]],[[2228.44,500,102.53],[3.82813E-9,0.707107,0.707107,-1.22165E-8],[1,0,2,0],[9E+9,9E+9,9E+9,9E+9,9E+9,9E+9]]],[[[1428.44,500,87.53],[3.82813E-9,0.707107,0.707107,-1.22165E-8],[1,0,2,0],[9E+9,9E+9,9E+9,9E+9,9E+9,9E+9]],[[1628.44,500,87.53],[3.82813E-9,0.707107,0.707107,-1.22165E-8],[1,0,2,0],[9E+9,9E+9,9E+9,9E+9,9E+9,9E+9]],[[1828.44,500,87.53],[3.82813E-9,0.707107,0.707107,-1.22165E-8],[1,0,2,0],[9E+9,9E+9,9E+9,9E+9,9E+9,9E+9]],[[2028.44,500,87.53],[3.82813E-9,0.707107,0.707107,-1.22165E-8],[1,0,2,0],[9E+9,9E+9,9E+9,9E+9,9E+9,9E+9]],[[2228.44,500,87.53],[3.82813E-9,0.707107,0.707107,-1.22165E-8],[1,0,2,0],[9E+9,9E+9,9E+9,9E+9,9E+9,9E+9]]],[[[1428.44,500,72.53],[3.82813E-9,0.707107,0.707107,-1.22165E-8],[1,0,2,0],[9E+9,9E+9,9E+9,9E+9,9E+9,9E+9]],[[1628.44,500,72.53],[3.82813E-9,0.707107,0.707107,-1.22165E-8],[1,0,2,0],[9E+9,9E+9,9E+9,9E+9,9E+9,9E+9]],[[1828.44,500,72.53],[3.82813E-9,0.707107,0.707107,-1.22165E-8],[1,0,2,0],[9E+9,9E+9,9E+9,9E+9,9E+9,9E+9]],[[2028.44,500,72.53],[3.82813E-9,0.707107,0.707107,-1.22165E-8],[1,0,2,0],[9E+9,9E+9,9E+9,9E+9,9E+9,9E+9]],[[2228.44,500,72.53],[3.82813E-9,0.707107,0.707107,-1.22165E-8],[1,0,2,0],[9E+9,9E+9,9E+9,9E+9,9E+9,9E+9]]],[[[1428.44,500,57.53],[3.82813E-9,0.707107,0.707107,-1.22165E-8],[1,0,2,0],[9E+9,9E+9,9E+9,9E+9,9E+9,9E+9]],[[1628.44,500,57.53],[3.82813E-9,0.707107,0.707107,-1.22165E-8],[1,0,2,0],[9E+9,9E+9,9E+9,9E+9,9E+9,9E+9]],[[1828.44,500,57.53],[3.82813E-9,0.707107,0.707107,-1.22165E-8],[1,0,2,0],[9E+9,9E+9,9E+9,9E+9,9E+9,9E+9]],[[2028.44,500,57.53],[3.82813E-9,0.707107,0.707107,-1.22165E-8],[1,0,2,0],[9E+9,9E+9,9E+9,9E+9,9E+9,9E+9]],[[2228.44,500,57.53],[3.82813E-9,0.707107,0.707107,-1.22165E-8],[1,0,2,0],[9E+9,9E+9,9E+9,9E+9,9E+9,9E+9]]],[[[1428.44,500,42.53],[3.82813E-9,0.707107,0.707107,-1.22165E-8],[1,0,2,0],[9E+9,9E+9,9E+9,9E+9,9E+9,9E+9]],[[1628.44,500,42.53],[3.82813E-9,0.707107,0.707107,-1.22165E-8],[1,0,2,0],[9E+9,9E+9,9E+9,9E+9,9E+9,9E+9]],[[1828.44,500,42.53],[3.82813E-9,0.707107,0.707107,-1.22165E-8],[1,0,2,0],[9E+9,9E+9,9E+9,9E+9,9E+9,9E+9]],[[2028.44,500,42.53],[3.82813E-9,0.707107,0.707107,-1.22165E-8],[1,0,2,0],[9E+9,9E+9,9E+9,9E+9,9E+9,9E+9]],[[2228.44,500,42.53],[3.82813E-9,0.707107,0.707107,-1.22165E-8],[1,0,2,0],[9E+9,9E+9,9E+9,9E+9,9E+9,9E+9]]],[[[1428.44,500,27.53],[3.82813E-9,0.707107,0.707107,-1.22165E-8],[1,0,2,0],[9E+9,9E+9,9E+9,9E+9,9E+9,9E+9]],[[1628.44,500,27.53],[3.82813E-9,0.707107,0.707107,-1.22165E-8],[1,0,2,0],[9E+9,9E+9,9E+9,9E+9,9E+9,9E+9]],[[1828.44,500,27.53],[3.82813E-9,0.707107,0.707107,-1.22165E-8],[1,0,2,0],[9E+9,9E+9,9E+9,9E+9,9E+9,9E+9]],[[2028.44,500,27.53],[3.82813E-9,0.707107,0.707107,-1.22165E-8],[1,0,2,0],[9E+9,9E+9,9E+9,9E+9,9E+9,9E+9]],[[2228.44,500,27.53],[3.82813E-9,0.707107,0.707107,-1.22165E-8],[1,0,2,0],[9E+9,9E+9,9E+9,9E+9,9E+9,9E+9]]],[[[1428.44,500,12.53],[3.82813E-9,0.707107,0.707107,-1.22165E-8],[1,0,2,0],[9E+9,9E+9,9E+9,9E+9,9E+9,9E+9]],[[1628.44,500,12.53],[3.82813E-9,0.707107,0.707107,-1.22165E-8],[1,0,2,0],[9E+9,9E+9,9E+9,9E+9,9E+9,9E+9]],[[1828.44,500,12.53],[3.82813E-9,0.707107,0.707107,-1.22165E-8],[1,0,2,0],[9E+9,9E+9,9E+9,9E+9,9E+9,9E+9]],[[2028.44,500,12.53],[3.82813E-9,0.707107,0.707107,-1.22165E-8],[1,0,2,0],[9E+9,9E+9,9E+9,9E+9,9E+9,9E+9]],[[2228.44,500,12.53],[3.82813E-9,0.707107,0.707107,-1.22165E-8],[1,0,2,0],[9E+9,9E+9,9E+9,9E+9,9E+9,9E+9]]]];
    PERS robtarget pPlace_work1_1:=[[749.06,1179.85,115.56],[4.15929E-07,8.35353E-07,-0.999897,-0.0143725],[0,0,-1,0],[9E+09,9E+09,9E+09,9E+09,9E+09,9E+09]];
    PERS robtarget pPlace_work1_2:=[[749.06,1103.50,115.56],[9.92289E-07,1.21612E-06,-0.999897,-0.014372],[0,0,-1,0],[9E+09,9E+09,9E+09,9E+09,9E+09,9E+09]];
    PERS robtarget pPlace_work1_3:=[[749.06,545.90,97.71],[9.15795E-07,9.05349E-07,-0.999897,-0.0143717],[0,1,-1,0],[9E+09,9E+09,9E+09,9E+09,9E+09,9E+09]];
    PERS robtarget pPlace_work1_4:=[[749.06,469.99,95.00],[1.15454E-06,9.965E-07,-0.999897,-0.0143717],[0,1,-1,0],[9E+09,9E+09,9E+09,9E+09,9E+09,9E+09]];
    PERS robtarget pPlace_work2_1:=[[749.06,344.27,104.21],[0.000956552,-0.999999,0.000961161,2.76734E-06],[-1,-1,2,0],[9E+09,9E+09,9E+09,9E+09,9E+09,9E+09]];
    PERS robtarget pPlace_work2_2:=[[749.06,420.58,105.25],[0.000956972,-1,1.18032E-05,2.48467E-06],[-1,-1,2,0],[9E+09,9E+09,9E+09,9E+09,9E+09,9E+09]];
    PERS robtarget pPlace_work2_3:=[[749.06,979.21,105.69],[0.000957149,-1,-6.73943E-05,2.25445E-06],[-1,-1,2,0],[9E+09,9E+09,9E+09,9E+09,9E+09,9E+09]];
    PERS robtarget pPlace_work2_4:=[[749.06,1055.75,107.07],[0.000957368,-1,-5.57621E-05,2.09476E-06],[-1,-2,2,0],[9E+09,9E+09,9E+09,9E+09,9E+09,9E+09]];
    PERS robtarget pPlace_work1_Panel_1:=[[1178.48,824.67,116.84],[0.00993253,-0.707036,-0.707038,-0.00993286],[0,0,0,0],[9E+09,9E+09,9E+09,9E+09,9E+09,9E+09]];
    PERS robtarget pPlace_work1_Panel_2:=[[1142.01,824.67,116.84],[0.00993252,-0.707036,-0.707038,-0.00993283],[0,0,0,0],[9E+09,9E+09,9E+09,9E+09,9E+09,9E+09]];
    PERS robtarget pPlace_work2_Panel_1:=[[1178.48,701.76,116.84],[0.000844486,-0.707106,-0.707107,-0.000843713],[-1,-1,1,0],[9E+09,9E+09,9E+09,9E+09,9E+09,9E+09]];
    PERS robtarget pPlace_work2_Panel_2:=[[1142.01,701.76,116.84],[0.000844498,-0.707106,-0.707107,-0.000843649],[-1,-1,1,0],[9E+09,9E+09,9E+09,9E+09,9E+09,9E+09]];
    PERS robtarget pPlace_work1_Panel_3:=[[628.48,824.67,116.84],[0.00993253,-0.707036,-0.707038,-0.00993286],[0,0,0,0],[9E+09,9E+09,9E+09,9E+09,9E+09,9E+09]];
    PERS robtarget pPlace_work1_Panel_4:=[[592.01,824.67,116.84],[0.00993252,-0.707036,-0.707038,-0.00993283],[0,0,0,0],[9E+09,9E+09,9E+09,9E+09,9E+09,9E+09]];
    PERS robtarget pPlace_work2_Panel_3:=[[628.48,701.76,116.84],[0.000844482,-0.707106,-0.707107,-0.000843775],[-1,-1,1,0],[9E+09,9E+09,9E+09,9E+09,9E+09,9E+09]];
    PERS robtarget pPlace_work2_Panel_4:=[[592.01,701.76,116.84],[0.000844431,-0.707106,-0.707107,-0.000843689],[-1,-1,1,0],[9E+09,9E+09,9E+09,9E+09,9E+09,9E+09]];
    PERS robtarget pPlace_work1_Panel_5:=[[305.29,824.67,116.84],[0.0099325,-0.707036,-0.707038,-0.00993282],[0,0,0,0],[9E+09,9E+09,9E+09,9E+09,9E+09,9E+09]];
    PERS robtarget pPlace_work2_Panel_5:=[[63.63,701.76,116.84],[0.000844667,-0.707106,-0.707106,-0.000843613],[-1,-2,1,0],[9E+09,9E+09,9E+09,9E+09,9E+09,9E+09]];
    PERS robtarget pPick_work1_Board:=[[609.44,824.67,116.84],[0.00993255,-0.707036,-0.707038,-0.0099329],[0,0,0,0],[9E+09,9E+09,9E+09,9E+09,9E+09,9E+09]];
    PERS robtarget pPick_work2_Board:=[[609.44,701.76,116.84],[0.000844469,-0.707106,-0.707107,-0.000843668],[-1,-1,1,0],[9E+09,9E+09,9E+09,9E+09,9E+09,9E+09]];
    PERS robtarget pPlace_Board_1:=[[1941.85,497.51,130.53],[2.40162E-08,0.707107,-0.707107,7.07584E-09],[-2,-1,-3,0],[9E+09,9E+09,9E+09,9E+09,9E+09,9E+09]];
    PERS robtarget pPlace_Board_2:=[[741.02,497.51,130.53],[2.66338E-08,0.707107,-0.707107,-1.17313E-09],[-2,-1,-3,0],[9E+09,9E+09,9E+09,9E+09,9E+09,9E+09]];
    PERS num Holder_Floor:=1;
    PERS num Holder_Count:=1;
    PERS num Panel_Floor:=5;
    PERS num Panel_Count:=1;
    PERS num Board_Floor:=3;
    PERS num Board_Count:=10;
    PERS bool LeftOK:=FALSE;
    PERS bool RightOK:=FALSE;
    PERS bool LeftPlaceOK:=TRUE;
    PERS bool RightPlaceOK:=TRUE;
    PERS bool LastPlaceOK:=false;
    CONST robtarget pMove_Holder_1:=[[1356.45,856.18,870.38],[1.27707E-07,-9.02504E-07,0.865853,0.500299],[0,0,-1,0],[9E+09,9E+09,9E+09,9E+09,9E+09,9E+09]];
    CONST robtarget pMove_Holder_2:=[[2588.00,142.39,881.49],[2.78546E-07,1.75287E-06,-0.865853,-0.500298],[0,1,-1,0],[9E+09,9E+09,9E+09,9E+09,9E+09,9E+09]];
    VAR robtarget pPlace_Board_Move{10,2}:=[[[[2201.66,-73.60,901.28],[7.27892E-09,-1.2141E-06,0.865853,0.500299],[0,0,0,0],[9E+09,9E+09,9E+09,9E+09,9E+09,9E+09]],[[2201.66,-73.60,901.28],[7.27892E-09,-1.2141E-06,0.865853,0.500299],[0,0,0,0],[9E+09,9E+09,9E+09,9E+09,9E+09,9E+09]]],[[[2201.66,-73.60,901.28],[7.27892E-09,-1.2141E-06,0.865853,0.500299],[0,0,0,0],[9E+09,9E+09,9E+09,9E+09,9E+09,9E+09]],[[2201.66,-73.60,901.28],[7.27892E-09,-1.2141E-06,0.865853,0.500299],[0,0,0,0],[9E+09,9E+09,9E+09,9E+09,9E+09,9E+09]]],[[[2201.66,-73.60,901.28],[7.27892E-09,-1.2141E-06,0.865853,0.500299],[0,0,0,0],[9E+09,9E+09,9E+09,9E+09,9E+09,9E+09]],[[2201.66,-73.60,901.28],[7.27892E-09,-1.2141E-06,0.865853,0.500299],[0,0,0,0],[9E+09,9E+09,9E+09,9E+09,9E+09,9E+09]]],[[[2201.66,-73.60,901.28],[7.27892E-09,-1.2141E-06,0.865853,0.500299],[0,0,0,0],[9E+09,9E+09,9E+09,9E+09,9E+09,9E+09]],[[2201.66,-73.60,901.28],[7.27892E-09,-1.2141E-06,0.865853,0.500299],[0,0,0,0],[9E+09,9E+09,9E+09,9E+09,9E+09,9E+09]]],[[[2201.66,-73.60,901.28],[7.27892E-09,-1.2141E-06,0.865853,0.500299],[0,0,0,0],[9E+09,9E+09,9E+09,9E+09,9E+09,9E+09]],[[2201.66,-73.60,901.28],[7.27892E-09,-1.2141E-06,0.865853,0.500299],[0,0,0,0],[9E+09,9E+09,9E+09,9E+09,9E+09,9E+09]]],[[[2201.66,-73.60,901.28],[7.27892E-09,-1.2141E-06,0.865853,0.500299],[0,0,0,0],[9E+09,9E+09,9E+09,9E+09,9E+09,9E+09]],[[2201.66,-73.60,901.28],[7.27892E-09,-1.2141E-06,0.865853,0.500299],[0,0,0,0],[9E+09,9E+09,9E+09,9E+09,9E+09,9E+09]]],[[[2201.66,-73.60,901.28],[7.27892E-09,-1.2141E-06,0.865853,0.500299],[0,0,0,0],[9E+09,9E+09,9E+09,9E+09,9E+09,9E+09]],[[2201.66,-73.60,901.28],[7.27892E-09,-1.2141E-06,0.865853,0.500299],[0,0,0,0],[9E+09,9E+09,9E+09,9E+09,9E+09,9E+09]]],[[[2201.66,-73.60,901.28],[7.27892E-09,-1.2141E-06,0.865853,0.500299],[0,0,0,0],[9E+09,9E+09,9E+09,9E+09,9E+09,9E+09]],[[2201.66,-73.60,901.28],[7.27892E-09,-1.2141E-06,0.865853,0.500299],[0,0,0,0],[9E+09,9E+09,9E+09,9E+09,9E+09,9E+09]]],[[[2201.66,-73.60,901.28],[7.27892E-09,-1.2141E-06,0.865853,0.500299],[0,0,0,0],[9E+09,9E+09,9E+09,9E+09,9E+09,9E+09]],[[2201.66,-73.60,901.28],[7.27892E-09,-1.2141E-06,0.865853,0.500299],[0,0,0,0],[9E+09,9E+09,9E+09,9E+09,9E+09,9E+09]]],[[[2201.66,-73.60,901.28],[7.27892E-09,-1.2141E-06,0.865853,0.500299],[0,0,0,0],[9E+09,9E+09,9E+09,9E+09,9E+09,9E+09]],[[2201.66,-73.60,901.28],[7.27892E-09,-1.2141E-06,0.865853,0.500299],[0,0,0,0],[9E+09,9E+09,9E+09,9E+09,9E+09,9E+09]]]];
    VAR intnum intno1:=0;
    VAR intnum intno2:=0;
    PERS robtarget pMove_1:=[[2411.98,-211.01,931.30],[7.28748E-08,-2.58327E-07,1,7.83697E-08],[0,-1,0,0],[9E+09,9E+09,9E+09,9E+09,9E+09,9E+09]];
    PERS robtarget pMove_2:=[[845.95,-0.00,932.98],[9.48304E-08,-0.707107,-0.707107,-4.28484E-08],[-1,0,0,0],[9E+09,9E+09,9E+09,9E+09,9E+09,9E+09]];
    PERS robtarget pMove_3:=[[-823.78,806.78,532.39],[5.50754E-07,6.36181E-07,-0.999897,-0.0143725],[1,-1,1,0],[9E+09,9E+09,9E+09,9E+09,9E+09,9E+09]];
    PERS robtarget pPlace_holder_1{4}:=[[[661.17,-0.00,932.98],[3.16101E-08,-0.707107,-0.707107,-7.01488E-10],[-1,0,1,0],[9E+09,9E+09,9E+09,9E+09,9E+09,9E+09]],[[661.17,-0.00,932.98],[3.16101E-08,-0.707107,-0.707107,-7.01488E-10],[-1,0,1,0],[9E+09,9E+09,9E+09,9E+09,9E+09,9E+09]],[[661.17,-0.00,932.98],[3.16101E-08,-0.707107,-0.707107,-7.01488E-10],[-1,0,1,0],[9E+09,9E+09,9E+09,9E+09,9E+09,9E+09]],[[661.17,-0.00,932.98],[3.16101E-08,-0.707107,-0.707107,-7.01488E-10],[-1,0,1,0],[9E+09,9E+09,9E+09,9E+09,9E+09,9E+09]]];
    PERS robtarget pPlace_holder_2{4}:=[[[661.17,-0.00,932.98],[3.16101E-08,-0.707107,-0.707107,-7.01488E-10],[-1,0,1,0],[9E+09,9E+09,9E+09,9E+09,9E+09,9E+09]],[[661.17,-0.00,932.98],[3.16101E-08,-0.707107,-0.707107,-7.01488E-10],[-1,0,1,0],[9E+09,9E+09,9E+09,9E+09,9E+09,9E+09]],[[661.17,-0.00,932.98],[3.16101E-08,-0.707107,-0.707107,-7.01488E-10],[-1,0,1,0],[9E+09,9E+09,9E+09,9E+09,9E+09,9E+09]],[[661.17,-0.00,932.98],[3.16101E-08,-0.707107,-0.707107,-7.01488E-10],[-1,0,1,0],[9E+09,9E+09,9E+09,9E+09,9E+09,9E+09]]];
    PERS robtarget pPlace_Panel_1{5}:=[[[661.17,-0.00,932.98],[3.16101E-08,-0.707107,-0.707107,-7.01488E-10],[-1,0,1,0],[9E+09,9E+09,9E+09,9E+09,9E+09,9E+09]],[[661.17,-0.00,932.98],[3.16101E-08,-0.707107,-0.707107,-7.01488E-10],[-1,0,1,0],[9E+09,9E+09,9E+09,9E+09,9E+09,9E+09]],[[661.17,-0.00,932.98],[3.16101E-08,-0.707107,-0.707107,-7.01488E-10],[-1,0,1,0],[9E+09,9E+09,9E+09,9E+09,9E+09,9E+09]],[[661.17,-0.00,932.98],[3.16101E-08,-0.707107,-0.707107,-7.01488E-10],[-1,0,1,0],[9E+09,9E+09,9E+09,9E+09,9E+09,9E+09]],[[661.17,-0.00,932.98],[3.16101E-08,-0.707107,-0.707107,-7.01488E-10],[-1,0,1,0],[9E+09,9E+09,9E+09,9E+09,9E+09,9E+09]]];
    PERS robtarget pPlace_Panel_2{5}:=[[[661.17,-0.00,932.98],[3.16101E-08,-0.707107,-0.707107,-7.01488E-10],[-1,0,1,0],[9E+09,9E+09,9E+09,9E+09,9E+09,9E+09]],[[661.17,-0.00,932.98],[3.16101E-08,-0.707107,-0.707107,-7.01488E-10],[-1,0,1,0],[9E+09,9E+09,9E+09,9E+09,9E+09,9E+09]],[[661.17,-0.00,932.98],[3.16101E-08,-0.707107,-0.707107,-7.01488E-10],[-1,0,1,0],[9E+09,9E+09,9E+09,9E+09,9E+09,9E+09]],[[661.17,-0.00,932.98],[3.16101E-08,-0.707107,-0.707107,-7.01488E-10],[-1,0,1,0],[9E+09,9E+09,9E+09,9E+09,9E+09,9E+09]],[[661.17,-0.00,932.98],[3.16101E-08,-0.707107,-0.707107,-7.01488E-10],[-1,0,1,0],[9E+09,9E+09,9E+09,9E+09,9E+09,9E+09]]];
    VAR pos pos1_Left:=[0,0,0];
    VAR pos pos1_Right:=[0,0,0];
    VAR shapedata shape1;
    VAR wztemporary wztemp1:=[0];
    VAR wzstationary wzstat1:=[0];
    VAR pos pos2_Left:=[0,0,0];
    VAR pos pos2_Right:=[0,0,0];
    VAR wzstationary wzstat2:=[0];
    VAR shapedata shape2;
    CONST robtarget pMove_4:=[[2936.69,1926.26,1288.99],[0.00337426,0.703346,0.710832,-0.00333845],[0,-1,1,0],[9E+09,9E+09,9E+09,9E+09,9E+09,9E+09]];
    CONST robtarget pMove_5:=[[2066.98,1304.72,1288.99],[0.000127656,0.999629,0.0268279,-0.00474495],[-1,-1,0,0],[9E+09,9E+09,9E+09,9E+09,9E+09,9E+09]];
    !***********************************************************
    !
    ! Module:  Module1
    !
    ! Description:
    !   <Insert description here>
    !
    ! Author: Administrator
    !
    ! Version: 1.0
    !
    !***********************************************************


    !***********************************************************
    !
    ! Procedure main
    !
    !   This is the entry point of your program
    !
    !***********************************************************
    PROC main()
        rResetAll;
        rCheckHomePos;
        WHILE TRUE DO
            IF LeftPlaceOK=FALSE THEN
                rLeft;
            ELSEIF RightPlaceOK=FALSE THEN
                rRight;
            ELSEIF LeftOK AND LeftPlaceOK THEN
                rLeftBoard;
            ELSEIF RightOK AND RightPlaceOK THEN
                rRightBoard;
            ENDIF
            rCheckHomePos;
            WaitTime 0.3;
        ENDWHILE
    ENDPROC

    PROC rResetAll()
        IDelete intno1;
        CONNECT intno1 WITH tLeft;
        ISignalDI Di03_LeftOK,1,intno1;
        IDelete intno2;
        CONNECT intno2 WITH tRight;
        ISignalDI Di04_RightOK,1,intno2;
        Reset Do01_Vacuum1;
        Reset Do02_Vacuum2;
        Reset Do03_LeftAllow;
        Reset Do04_RightAllow;
        Reset Do05_RawEmpty;
        Reset Do06_FinishFull;
        rCount;
        Holder_Floor:=1;
        Holder_Count:=1;
        Panel_Floor:=1;
        Panel_Count:=1;
        LeftOK:=FALSE;
        RightOK:=FALSE;
        LeftPlaceOK:=FALSE;
        RightPlaceOK:=FALSE;
        LastPlaceOK:=FALSE;
    ENDPROC

    PROC rCheckHomePos()
        VAR robtarget pActualPos;
        IF NOT CurrentPos(pHome,Tool_Vacuum) THEN
            pActualPos:=CRobT(\Tool:=Tool_Vacuum\WObj:=wobj0);
            pActualPos.trans.z:=pHome.trans.z+100;
            MoveL pActualPos,v200,z10,Tool_Vacuum;
            MoveJ pHome,v1000,fine,Tool_Vacuum;
        ENDIF
    ENDPROC

    FUNC bool CurrentPos(robtarget ComparePos,INOUT tooldata TCP)
        VAR num Counter:=0;
        VAR robtarget ActualPos;
        ActualPos:=CRobT(\Tool:=TCP\WObj:=wobj0);
        IF ActualPos.trans.x>ComparePos.trans.x-200 AND ActualPos.trans.x<ComparePos.trans.x+200 Counter:=Counter+1;
        IF ActualPos.trans.y>ComparePos.trans.y-200 AND ActualPos.trans.y<ComparePos.trans.y+200 Counter:=Counter+1;
        IF ActualPos.trans.z>ComparePos.trans.z-100 AND ActualPos.trans.z<ComparePos.trans.z+100 Counter:=Counter+1;
        IF ActualPos.rot.q1>ComparePos.rot.q1-0.1 AND ActualPos.rot.q1<ComparePos.rot.q1+0.1 Counter:=Counter+1;
        IF ActualPos.rot.q2>ComparePos.rot.q2-0.1 AND ActualPos.rot.q2<ComparePos.rot.q2+0.1 Counter:=Counter+1;
        IF ActualPos.rot.q3>ComparePos.rot.q3-0.1 AND ActualPos.rot.q3<ComparePos.rot.q3+0.1 Counter:=Counter+1;
        IF ActualPos.rot.q4>ComparePos.rot.q4-0.1 AND ActualPos.rot.q4<ComparePos.rot.q4+0.1 Counter:=Counter+1;
        RETURN Counter=7;
    ENDFUNC

    PROC rLeft()
        rPick_Holder;
        rPlace pPlace_work1_1,pPlace_work1_2,Wobj_Left;
        rPick_Holder;
        rPlace pPlace_work1_3,pPlace_work1_4,Wobj_Left;
        rPick_Panel;
        rPlace pPlace_work1_Panel_1,pPlace_work1_Panel_2,Wobj_Left;
        rPick_Panel;
        rPlace pPlace_work1_Panel_3,pPlace_work1_Panel_4,Wobj_Left;
        rLeft_Panel_5;
        LeftPlaceOK:=TRUE;
        Set Do03_LeftAllow;
    ENDPROC

    PROC rRight()
        rPick_Holder;
        MoveJ pMove_2,v1000,z50,tool0;
        rPlace pPlace_work2_1,pPlace_work2_2,Wobj_Right;
        rPick_Holder;
        MoveJ pMove_2,v1000,z50,tool0;
        rPlace pPlace_work2_3,pPlace_work2_4,Wobj_Right;
        rPick_Panel;
        MoveJ pMove_2,v1000,z50,tool0;
        rPlace pPlace_work2_Panel_1,pPlace_work2_Panel_2,Wobj_Right;
        rPick_Panel;
        MoveJ pMove_2,v1000,z50,tool0;
        rPlace pPlace_work2_Panel_3,pPlace_work2_Panel_4,Wobj_Right;
        rRight_Panel_5;
        RightPlaceOK:=TRUE;
        Set Do04_RightAllow;
    ENDPROC

    PROC rLeftBoard()
        LeftOK:=FALSE;
        LeftPlaceOK:=FALSE;
        rPick_Board pPick_work1_Board,Wobj_Left;
        rPlace_Board;
    ENDPROC

    PROC rRightBoard()
        RightOK:=FALSE;
        RightPlaceOK:=FALSE;
        rPick_Board pPick_work2_Board,Wobj_Right;
        rPlace_Board;
    ENDPROC

    PROC rLeft_Panel_5()
        MoveL pMove_1,v2000,z10,Tool_Vacuum\WObj:=Wobj_materials;
        MoveJ offs(pPick_Panel_Move1{Panel_Floor,3},0,0,200),v2000,z10,Tool_Vacuum\WObj:=Wobj_materials;
        MoveJ pPick_Panel_Move1{Panel_Floor,3},v2000,fine,Tool_Vacuum\WObj:=Wobj_materials;
        Set Do01_Vacuum1;
        WaitTime 0.3;
        MoveJ offs(pPick_Panel_Move1{Panel_Floor,3},0,0,200),v2000,z10,Tool_Vacuum\WObj:=Wobj_materials;
        MoveL pMove_1,v2000,z10,Tool_Vacuum\WObj:=Wobj_materials;
        MoveJ Offs(pPlace_work1_Panel_5,0,0,200),v2000,z10,Tool_Vacuum\WObj:=Wobj_Left;
        MoveJ pPlace_work1_Panel_5,v2000,fine,Tool_Vacuum\WObj:=Wobj_Left;
        Reset Do01_Vacuum1;
        WaitTime 0.3;
        MoveJ Offs(pPlace_work1_Panel_5,0,0,100),v2000,z10,Tool_Vacuum\WObj:=Wobj_Left;
    ENDPROC

    PROC rRight_Panel_5()
        MoveL pMove_1,v2000,z10,Tool_Vacuum\WObj:=Wobj_materials;
        MoveJ offs(pPick_Panel_Move2{Panel_Floor,3},0,0,200),v2000,z10,Tool_Vacuum\WObj:=Wobj_materials;
        MoveJ pPick_Panel_Move2{Panel_Floor,3},v2000,fine,Tool_Vacuum\WObj:=Wobj_materials;
        Set Do02_Vacuum2;
        WaitTime 0.3;
        MoveJ offs(pPick_Panel_Move2{Panel_Floor,3},0,0,200),v2000,z10,Tool_Vacuum\WObj:=Wobj_materials;
        MoveL pMove_1,v2000,z10,Tool_Vacuum\WObj:=Wobj_materials;
        MoveL pMove_2,v2000,z10,Tool_Vacuum\WObj:=wobj0;
        MoveJ Offs(pPlace_work2_Panel_5,0,0,100),v2000,z10,Tool_Vacuum\WObj:=Wobj_Right;
        MoveJ pPlace_work2_Panel_5,v2000,fine,Tool_Vacuum\WObj:=Wobj_Right;
        Reset Do02_Vacuum2;
        WaitTime 0.3;
        MoveJ Offs(pPlace_work2_Panel_5,0,0,200),v2000,z10,Tool_Vacuum\WObj:=Wobj_Right;
    ENDPROC

    PROC rPick_Holder()
        MoveJ pMove_1,v2000,z10,Tool_Vacuum\WObj:=Wobj_materials;
        MoveJ offs(pPick_holder_Move1{Holder_Floor,Holder_Count},0,0,200),v2000,z10,Tool_Vacuum\WObj:=Wobj_materials;
        MoveJ pPick_holder_Move1{Holder_Floor,Holder_Count},v2000,fine,Tool_Vacuum\WObj:=Wobj_materials;
        Set Do01_Vacuum1;
        WaitTime 0.3;
        MoveJ offs(pPick_holder_Move1{Holder_Floor,Holder_Count},0,0,200),v2000,z10,Tool_Vacuum\WObj:=Wobj_materials;
        MoveJ offs(pPick_holder_Move2{Holder_Floor,Holder_Count},0,0,200),v2000,z10,Tool_Vacuum\WObj:=Wobj_materials;
        MoveJ pPick_holder_Move2{Holder_Floor,Holder_Count},v2000,fine,Tool_Vacuum\WObj:=Wobj_materials;
        Set Do02_Vacuum2;
        WaitTime 0.3;
        MoveJ offs(pPick_holder_Move2{Holder_Floor,Holder_Count},0,0,200),v2000,z10,Tool_Vacuum\WObj:=Wobj_materials;
        Incr Holder_Count;
        IF Holder_Count>=11 THEN
            Incr Holder_Floor;
            Holder_Count:=1;
        ENDIF
        IF Holder_Floor>=5 THEN
            Holder_Floor:=1;
            Holder_Count:=1;
        ENDIF
        MoveJ pMove_1,v2000,z10,Tool_Vacuum\WObj:=Wobj_materials;
    ENDPROC

    PROC rPick_Panel()
        MoveL pMove_1,v2000,z10,Tool_Vacuum\WObj:=Wobj_materials;
        MoveJ offs(pPick_Panel_Move1{Panel_Floor,Panel_Count},0,0,200),v2000,z10,Tool_Vacuum\WObj:=Wobj_materials;
        MoveJ pPick_Panel_Move1{Panel_Floor,Panel_Count},v2000,fine,Tool_Vacuum\WObj:=Wobj_materials;
        Set Do01_Vacuum1;
        WaitTime 0.3;
        MoveJ offs(pPick_Panel_Move1{Panel_Floor,Panel_Count},0,0,200),v2000,z10,Tool_Vacuum\WObj:=Wobj_materials;
        MoveJ offs(pPick_Panel_Move2{Panel_Floor,Panel_Count},0,0,200),v2000,z10,Tool_Vacuum\WObj:=Wobj_materials;
        MoveJ pPick_Panel_Move2{Panel_Floor,Panel_Count},v2000,fine,Tool_Vacuum\WObj:=Wobj_materials;
        Set Do02_Vacuum2;
        WaitTime 0.3;
        MoveJ offs(pPick_Panel_Move2{Panel_Floor,Panel_Count},0,0,200),v2000,z10,Tool_Vacuum\WObj:=Wobj_materials;
        Incr Panel_Count;
        IF Panel_Count>=6 THEN
            Incr Panel_Floor;
            Panel_Count:=1;
        ENDIF
        IF Panel_Count=3 THEN
            Incr Panel_Count;
        ENDIF
        IF Panel_Floor>=21 THEN
            Panel_Floor:=1;
            Panel_Count:=1;
        ENDIF
        MoveJ [[2401.26,95.18,814.51],[0.321953,-0.629561,-0.62956,-0.321953],[0,1,0,0],[9E+09,9E+09,9E+09,9E+09,9E+09,9E+09]],v2000,z10,Tool_Vacuum\WObj:=Wobj_materials;
    ENDPROC

    PROC rPoint()
        MoveJ pPick_holder_1,v1000,fine,Tool_Vacuum\WObj:=Wobj_materials;
        MoveJ pPick_holder_2,v1000,fine,Tool_Vacuum\WObj:=Wobj_materials;
        MoveJ pPick_Panel_1,v1000,fine,Tool_Vacuum\WObj:=Wobj_materials;
        MoveJ pPick_Panel_2,v1000,fine,Tool_Vacuum\WObj:=Wobj_materials;
        MoveJ pPlace_work1_1,v1000,fine,Tool_Vacuum\WObj:=Wobj_Left;
        MoveJ pPlace_work1_2,v1000,fine,Tool_Vacuum\WObj:=Wobj_Left;
        MoveJ pPlace_work1_3,v1000,fine,Tool_Vacuum\WObj:=Wobj_Left;
        MoveJ pPlace_work1_4,v1000,fine,Tool_Vacuum\WObj:=Wobj_Left;
        MoveJ pPlace_work2_1,v1000,fine,Tool_Vacuum\WObj:=Wobj_Right;
        MoveJ pPlace_work2_2,v1000,fine,Tool_Vacuum\WObj:=Wobj_Right;
        MoveJ pPlace_work2_3,v1000,fine,Tool_Vacuum\WObj:=Wobj_Right;
        MoveJ pPlace_work2_4,v1000,fine,Tool_Vacuum\WObj:=Wobj_Right;
        MoveJ pPlace_work1_Panel_1,v1000,fine,Tool_Vacuum\WObj:=Wobj_Left;
        MoveJ pPlace_work1_Panel_2,v1000,fine,Tool_Vacuum\WObj:=Wobj_Left;
        MoveJ pPlace_work1_Panel_3,v1000,fine,Tool_Vacuum\WObj:=Wobj_Left;
        MoveJ pPlace_work1_Panel_4,v1000,fine,Tool_Vacuum\WObj:=Wobj_Left;
        MoveJ pPlace_work1_Panel_5,v1000,fine,Tool_Vacuum\WObj:=Wobj_Left;
        MoveJ pPlace_work2_Panel_1,v1000,fine,Tool_Vacuum\WObj:=Wobj_Right;
        MoveJ pPlace_work2_Panel_2,v1000,fine,Tool_Vacuum\WObj:=Wobj_Right;
        MoveJ pPlace_work2_Panel_3,v1000,fine,Tool_Vacuum\WObj:=Wobj_Right;
        MoveJ pPlace_work2_Panel_4,v1000,fine,Tool_Vacuum\WObj:=Wobj_Right;
        MoveJ pPlace_work2_Panel_5,v1000,fine,Tool_Vacuum\WObj:=Wobj_Right;
        MoveJ pPick_work1_Board,v1000,fine,Tool_Vacuum\WObj:=Wobj_Left;
        MoveJ pPick_work2_Board,v1000,fine,Tool_Vacuum\WObj:=Wobj_Right;
        MoveJ pPlace_Board_1,v1000,fine,Tool_Vacuum\WObj:=Wobj_Board;
        MoveJ pPlace_Board_2,v1000,fine,Tool_Vacuum\WObj:=Wobj_Board;
    ENDPROC

    PROC rCount()
        FOR i FROM 1 TO 4 DO
            FOR j FROM 1 TO 10 DO
                pPick_Holder_Move1{i,j}:=Offs(pPick_holder_1,0,100*(j-1),-120*(i-1));
            ENDFOR
        ENDFOR
        FOR i FROM 1 TO 4 DO
            FOR j FROM 1 TO 10 DO
                pPick_Holder_Move2{i,j}:=Offs(pPick_holder_2,0,100*(j-1),-120*(i-1));
            ENDFOR
        ENDFOR
        FOR i FROM 1 TO 20 DO
            FOR j FROM 1 TO 5 DO
                pPick_Panel_Move1{i,j}:=Offs(pPick_Panel_1,200*(j-1),0,-15*(i-1));
            ENDFOR
        ENDFOR
        FOR i FROM 1 TO 20 DO
            FOR j FROM 1 TO 5 DO
                pPick_Panel_Move2{i,j}:=Offs(pPick_Panel_2,200*(j-1),0,-15*(i-1));
            ENDFOR
        ENDFOR
        FOR i FROM 1 TO 10 DO
            FOR j FROM 1 TO 2 DO
                pPlace_Board_Move{i,j}:=Offs(pPlace_Board_2,1200*(j-1),0,135*(i-1));
            ENDFOR
        ENDFOR
    ENDPROC

    PROC rPlace(robtarget point1,robtarget point2,INOUT wobjdata Wobj)
        MoveL Offs(point1,0,0,400),v2000,z10,Tool_Vacuum\WObj:=Wobj;
        MoveJ Point1,v2000,fine,Tool_Vacuum\WObj:=Wobj;
        Reset Do02_Vacuum2;
        WaitTime 0.3;
        MoveJ Offs(point1,0,0,20),v2000,z10,Tool_Vacuum\WObj:=Wobj;
        MoveJ Offs(point2,0,0,20),v2000,z10,Tool_Vacuum\WObj:=Wobj;
        MoveJ Point2,v2000,fine,Tool_Vacuum\WObj:=Wobj;
        Reset Do01_Vacuum1;
        WaitTime 0.3;
        MoveJ offs(Point2,0,0,200),v2000,z10,Tool_Vacuum\WObj:=Wobj;
    ENDPROC

    PROC rPick_Board(robtarget point1,INOUT wobjdata wobj)
        MoveJ offs(Point1,0,0,200),v2000,z10,Tool_Vacuum\WObj:=Wobj;
        MoveJ Point1,v2000,fine,Tool_Vacuum\WObj:=Wobj;
        Set Do01_Vacuum1;
        Set Do02_Vacuum2;
        WaitTime 0.3;
        MoveJ Offs(point1,0,0,200),v2000,z10,Tool_Vacuum\WObj:=Wobj;
    ENDPROC

    PROC rPlace_Board()
        MoveJ pMove_4, v1000, z10, Tool_Vacuum\WObj:=Wobj_Board;
        MoveJ pMove_5, v1000, z10, Tool_Vacuum\WObj:=Wobj_Board;
        MoveJ Offs(pPlace_Board_Move{Board_Floor,Board_Count},0,0,200),v2000,z10,Tool_Vacuum\WObj:=Wobj_Board;
        MoveJ pPlace_Board_Move{Board_Floor,Board_Count},v2000,fine,Tool_Vacuum\WObj:=Wobj_Board;
        Reset Do01_Vacuum1;
        Reset Do02_Vacuum2;
        WaitTime 0.3;
        MoveJ offs(pPlace_Board_Move{Board_Floor,Board_Count},0,0,200),v2000,z10,Tool_Vacuum\WObj:=Wobj_Board;
        Incr Board_Count;
        IF Board_Count>=3 THEN
            Incr Board_Floor;
            Board_Count:=1;
        ENDIF
        IF Board_Floor>=11 THEN
            Board_Floor:=1;
            Board_Count:=1;
        ENDIF
    ENDPROC

    TRAP tLeft
        LeftOK:=TRUE;
        Reset Do03_LeftAllow;
    ENDTRAP

    TRAP tRight
        RightOK:=TRUE;
        Reset Do04_RightAllow;
    ENDTRAP

    PROC rSafe()
        pos1_Left:=[875,914,-50];
        pos2_Left:=[1900,1800,1400];
        WZBoxDef\Inside,shape1,pos1_Left,pos2_Left;
        WZDOSet\Stat,wzstat1\Inside,shape1,Do07_LeftSafeOut,0;
        pos1_Right:=[775,-845,-60];
        pos2_Right:=[1800,-1700,800];
        WZBoxDef\Inside,shape2,pos1_Right,pos2_Right;
        WZDOSet\Stat,wzstat2\Inside,shape2,Do08_RightSafeOut,0;
    ENDPROC
ENDMODULE
